PROGRAM MAIN
VAR
END_VAR

A_Program();

END_PROGRAM

(* stored: Version 1.1.0.1, ProductVersion 3.1.4025.12
   POU MAIN: Id {a6bb2f7f-8491-400d-8e97-78fbace84f29}, SpecialFunc None *)
